{attribute 'conditionalshow'}
FUNCTION_BLOCK FB_GantryXYZ EXTENDS FB_PackML_BaseModule
VAR
    // Sub module definitions here
	RecipeBuilder	:FB_RecipeBuilderWings;

	
	// List of sub modules
    ipSubModules_Init : ARRAY[1..Parameters_PackML_Base.MAX_NO_OF_SUBMODULES] OF I_PackML_BaseModule := [];

    // Component definitions here
    AxisX : FB_Component_BasicAxis := (Name := 'AxisX');
    AxisY : FB_Component_BasicAxis := (Name := 'AxisY');
    AxisZ : FB_Component_BasicAxis := (Name := 'AxisZ');
    CylinderCuttingY : FB_CylinderCutY := (Name := 'Cylinder Y');
	CylinderCuttingX : FB_CylinderCutX := (Name := 'Cylinder X');
	

    // Alarms for this module
    GantryAlarms : ARRAY[1..GANTRY_ALARM_COUNT] OF FB_TcAlarm;
	
    // Properties
    _HomingStepX :			INT;
    _HomingStepY :			INT;
    _HomingStepZ :			INT;

	_ProgramIdRequested :   E_RecipeID;
	_CurrentSpeed: 			LREAL;
	
	//Segments
	SegmentGrooves       : ARRAY[1..32] OF ST_CutSegment;
    SegmentsToGroove     : INT;          // Ile odcinków
    iSegmentsToGroove    : INT;          // Indeks aktualnego odcinka
    
    
	//Segments Cut Y
	SegmentCutY      	 : ARRAY[1..32] OF ST_CutSegment;
    SegmentsToCutY       : INT;          // Ile odcinków
    iSegmentsToCutY      : INT;          // Indeks aktualnego odcinka
	
	//Segments Cut X
	SegmentCutX      	 : ARRAY[1..32] OF ST_CutSegment;
    SegmentsToCutX       : INT;          // Ile odcinków
    iSegmentsToCutX      : INT;          // Indeks aktualnego odcinka

	//Sequencers
	OrchestratorStep :			INT := 0;
	ExecutorStep :				INT := 0;
	
	GantryXYZ_HMI : ST_GantryXYZ_HMI;
	
	//Test
	fbHomeStratX : FB_Homing_StandardNC;
    fbHomeStratY : FB_Homing_StandardNC;
    fbHomeStratZ : FB_Homing_StandardNC;
	
END_VAR

VAR PERSISTENT
	_CuttingSpeedX			:REAL;
	_CuttingSpeedY			:REAL;
	_CuttingIdleTime		:REAL;
	_CuttingOverpass		:REAL;
	_CutterXOffsetX			:REAL;
	_CutterXOffsetY			:REAL;
	_CutterYOffsetX			:REAL;
	_CutterYOffsetY			:REAL;	
    _GrooveDepthZ 			:REAL;
	_GroovingSpeedX 		:REAL;
	_GroovingSpeedY 		:REAL;
	_GroovingSpeedZ 		:REAL;
	_GroovingIdleTime 		:REAL;
    _GroovingOverpass 		:REAL;
    _PanelFrontWidth 		:REAL;
    _PanelHeight 			:REAL;
    _RailHeightCorrection	:REAL;
    _RapidSpeedX 			:REAL;
    _RapidSpeedY 			:REAL;
    _RapidSpeedZ 			:REAL;
	_GlobalOffset 			:INT;
END_VAR

VAR CONSTANT
    GANTRY_ALARM_COUNT : 	INT := 5;
END_VAR


METHOD PROTECTED Aborting
VAR
	i				: UDINT;
	SubModulesReady : BOOL := TRUE;
END_VAR
CASE _CurrentMode OF

	//=================================PRODUCTION MODE==================================
	E_PMLUnitMode.ePMLUnitMode_Production:
CASE SequenceState OF
    0:
        NoStateTasksToComplete := FALSE;
        SequenceState          := SequenceState + 10;
    10:
		AxisX.Disable();
		AxisY.Disable();
		AxisZ.Disable();

		IO.SpindleEnable := FALSE;
		IO.CoolingEnable := FALSE;
		
		CylinderCuttingX.Retract();
		CylinderCuttingY.Retract();

		THIS^.HomingStepX := 0;
		THIS^.HomingStepY := 0;
		THIS^.HomingStepZ := 0;
		OrchestratorStep := 0;
		ExecutorStep := 0;
		
		//test
		fbHomeStratX.Abort();
        fbHomeStratY.Abort();
        fbHomeStratZ.Abort();
		
		SequenceState := SequenceState + 10;
		
		
	20:

		StateTasksComplete := TRUE;
		SUPER^.Aborting();
END_CASE

	//=================================MAINTENANCE & MANUAL MODE==================================
	E_PMLUnitMode.ePMLUnitMode_Maintenance, E_PMLUnitMode.ePMLUnitMode_Manual:

	CASE SequenceState OF
    
	0:
        NoStateTasksToComplete := FALSE;
        SequenceState          := SequenceState + 10;
    
	10:
		AxisX.Disable();
		AxisY.Disable();
		AxisZ.Disable();
		
		IO.CoolingEnable := FALSE;
		IO.SpindleEnable := FALSE;
		THIS^.HomingStepX := 0;
		THIS^.HomingStepY := 0;
		THIS^.HomingStepZ := 0;
		OrchestratorStep := 0;
		SequenceState := SequenceState + 10;
	
	20:
		StateTasksComplete := TRUE;
		SUPER^.Aborting();
	END_CASE
	

	END_CASE
END_METHOD

METHOD BuildSegments_Arona : BOOL
//  Start → Stop, Milling Segments
SegmentsToGroove := 4;

SegmentGrooves[1].Start.X := 500;
SegmentGrooves[1].Start.Y := 500;
SegmentGrooves[1].Stop.X  := 0;
SegmentGrooves[1].Stop.Y  := 500;

SegmentGrooves[2].Start.X := 500;
SegmentGrooves[2].Start.Y := 0;
SegmentGrooves[2].Stop.X  := 0; 
SegmentGrooves[2].Stop.Y  := 0;

SegmentGrooves[3].Start.X := 500;
SegmentGrooves[3].Start.Y := 500;
SegmentGrooves[3].Stop.X  := 500;
SegmentGrooves[3].Stop.Y  := 0;

SegmentGrooves[4].Start.X := 0;
SegmentGrooves[4].Start.Y := 500;
SegmentGrooves[4].Stop.X  := 0;
SegmentGrooves[4].Stop.Y  := 0;

//  Start → Stop, CutY Segments
SegmentsToCutY := 2;

SegmentCutY[1].Start.X := 0; 
SegmentCutY[1].Start.Y := 500;  
SegmentCutY[1].Stop.X  := 0; 
SegmentCutY[1].Stop.Y  := 0;
SegmentCutY[2].Start.X := 500; 
SegmentCutY[2].Start.Y := 500;  
SegmentCutY[2].Stop.X  := 500; 
SegmentCutY[2].Stop.Y  := 0;

SegmentsToCutX := 2;

SegmentCutX[1].Start.X := 500; 
SegmentCutX[1].Start.Y := 500;  
SegmentCutX[1].Stop.X  := 500; 
SegmentCutX[1].Stop.Y  := 0;
SegmentCutX[2].Start.X := 0; 
SegmentCutX[2].Start.Y := 500;  
SegmentCutX[2].Stop.X  := 0; 
SegmentCutX[2].Stop.Y  := 0;



BuildSegments_Arona := TRUE;
END_METHOD

METHOD BuildSegments_BorgoFlaps : BOOL
VAR_INST
	TotalY 		:REAL;
	TotalX  	:REAL;
	ShorterY  	:REAL;
	ShorterX  	:REAL;
END_VAR
//Natural language parameters;
//TotalY := PanelFrontLength + 2 * _PanelHeight;
TotalX := PanelFrontWidth + 2 * _PanelHeight;
ShorterY := TotalY - _PanelHeight;
ShorterX := TotalX - _PanelHeight;


SegmentsToGroove := 4;

///////////////
SegmentGrooves[1].Start.X := TotalX;
SegmentGrooves[1].Stop.X := 0;

SegmentGrooves[1].Start.Y := ShorterY;
SegmentGrooves[1].Stop.Y := ShorterY;

/////////////
SegmentGrooves[2].Start.Y := TotalY;
SegmentGrooves[2].Stop.Y := 0;

SegmentGrooves[2].Start.X := _PanelHeight;
SegmentGrooves[2].Stop.X := _PanelHeight;

///////////////
SegmentGrooves[3].Start.X := 0;
SegmentGrooves[3].Stop.X :=  TotalX; 

SegmentGrooves[3].Start.Y := _PanelHeight;
SegmentGrooves[3].Stop.Y :=  _PanelHeight;

//////////////
SegmentGrooves[4].Start.X := ShorterX;
SegmentGrooves[4].Stop.X := ShorterX;

SegmentGrooves[4].Start.Y := 0;
SegmentGrooves[4].Stop.Y := TotalY;





//  Start → Stop, CutY Segments
SegmentsToCutY := 0;

SegmentsToCutX := 0;

BuildSegments_BorgoFlaps := TRUE;
END_METHOD

METHOD BuildSegments_BorgoWings : BOOL
VAR_INST
	TotalY 		:REAL;
	TotalX  	:REAL;
	ShorterY  	:REAL;
	ShorterX  	:REAL;
END_VAR

//We cut here BorgoWings it means, panel will be installed on wings
// It means we have to make flaps shorter
//Natural language parameters;
//TotalY := PanelFrontLength + 2 * _PanelHeight;
TotalX := PanelFrontWidth + 2 * _PanelHeight;
ShorterY := TotalY - _PanelHeight;
ShorterX := TotalX - _PanelHeight;



//  Start → Stop, Milling Segments
SegmentsToGroove := 4;

///////////////
SegmentGrooves[1].Start.X := TotalX;
SegmentGrooves[1].Stop.X := 0;

SegmentGrooves[1].Start.Y := ShorterY;
SegmentGrooves[1].Stop.Y := ShorterY;

///////////////
SegmentGrooves[2].Start.X := TotalX;
SegmentGrooves[2].Stop.X :=  0; 

SegmentGrooves[2].Start.Y := _PanelHeight;
SegmentGrooves[2].Stop.Y :=  _PanelHeight;

//////////////
SegmentGrooves[3].Start.X := ShorterX;
SegmentGrooves[3].Stop.X := ShorterX;

SegmentGrooves[3].Start.Y := TotalY;
SegmentGrooves[3].Stop.Y := 0;

/////////////
SegmentGrooves[4].Start.Y := TotalY;
SegmentGrooves[4].Stop.Y := 0;

SegmentGrooves[4].Start.X := _PanelHeight;
SegmentGrooves[4].Stop.X := _PanelHeight;


////////////
// Cut X //
///////////
SegmentsToCutX := 6;

//Short Box Segments
SegmentCutX[1].Start.X := TotalX + _CuttingOverpass;
SegmentCutX[1].Stop.X  := ShorterX;

SegmentCutX[1].Start.Y := ShorterY;
SegmentCutX[1].Stop.Y  := ShorterY;

///////////////
SegmentCutX[2].Start.X := _PanelHeight;
SegmentCutX[2].Stop.X  := -_CuttingOverpass;

SegmentCutX[2].Start.Y := ShorterY;
SegmentCutX[2].Stop.Y  := ShorterY;

///////////////
SegmentCutX[3].Start.X := TotalX + _CuttingOverpass;
SegmentCutX[3].Stop.X := ShorterX;

SegmentCutX[3].Start.Y := _PanelHeight;
SegmentCutX[3].Stop.Y := _PanelHeight;

///////////////
SegmentCutX[4].Start.X := _PanelHeight;
SegmentCutX[4].Stop.X :=  -_CuttingOverpass;

SegmentCutX[4].Start.Y := _PanelHeight;
SegmentCutX[4].Stop.Y := _PanelHeight;

//Panel Dimensions Shorter Flaps


SegmentCutX[5].Start.X := TotalX + _CuttingOverpass;
SegmentCutX[5].Stop.X  := - _CuttingOverpass;

SegmentCutX[5].Start.Y := TotalY - _RailHeightCorrection;
SegmentCutX[5].Stop.Y  := TotalY - _RailHeightCorrection;

///////////////
SegmentCutX[6].Start.X := TotalX + _CuttingOverpass;
SegmentCutX[6].Stop.X  := - _CuttingOverpass;

SegmentCutX[6].Start.Y := _RailHeightCorrection;
SegmentCutX[6].Stop.Y  := _RailHeightCorrection;


////////////
// Cut Y //
///////////

SegmentsToCutY := 6;

//Short Box Segments
SegmentCutY[1].Start.X := ShorterX;
SegmentCutY[1].Stop.X  := ShorterX;

SegmentCutY[1].Start.Y := TotalY + _CuttingOverpass;
SegmentCutY[1].Stop.Y  := ShorterY;

///////////////
SegmentCutY[2].Start.X := _PanelHeight;
SegmentCutY[2].Stop.X  := _PanelHeight;

SegmentCutY[2].Start.Y := TotalY + _CuttingOverpass;
SegmentCutY[2].Stop.Y  := ShorterY;

///////////////
SegmentCutY[3].Start.X := ShorterX;
SegmentCutY[3].Stop.X  := ShorterX;

SegmentCutY[3].Start.Y := _PanelHeight;
SegmentCutY[3].Stop.Y  := -_CuttingOverpass;

///////////////
SegmentCutY[4].Start.X := _PanelHeight;
SegmentCutY[4].Stop.X  := _PanelHeight;

SegmentCutY[4].Start.Y := _PanelHeight;
SegmentCutY[4].Stop.Y  := -_CuttingOverpass;

//Panel Dimensions
SegmentCutY[5].Start.X := TotalX;
SegmentCutY[5].Stop.X  := TotalX;

SegmentCutY[5].Start.Y := TotalY + _CuttingOverpass;
SegmentCutY[5].Stop.Y  := -_CuttingOverpass;
///////////////
SegmentCutY[6].Start.X := 0;
SegmentCutY[6].Stop.X  := 0;

SegmentCutY[6].Start.Y := TotalY + _CuttingOverpass;
SegmentCutY[6].Stop.Y  := - _CuttingOverpass;



BuildSegments_BorgoWings := TRUE;
END_METHOD

METHOD BuildSegments_Calibration : BOOL
VAR_INST
	TotalLength :REAL;
	TotalWidth  :REAL;
	WingHeight  :REAL;
	FlapHeight  :REAL;
END_VAR
//  Start → Stop, Milling Segments
SegmentsToGroove := 4;

SegmentGrooves[1].Start.X := 300;
SegmentGrooves[1].Start.Y := 300;
SegmentGrooves[1].Stop.X  := 50;
SegmentGrooves[1].Stop.Y  := 300;

SegmentGrooves[2].Start.X := 300;
SegmentGrooves[2].Start.Y := 50;
SegmentGrooves[2].Stop.X  := 50; 
SegmentGrooves[2].Stop.Y  := 50;

SegmentGrooves[3].Start.X := 300;
SegmentGrooves[3].Start.Y := 300;
SegmentGrooves[3].Stop.X  := 300;
SegmentGrooves[3].Stop.Y  := 50;

SegmentGrooves[4].Start.X := 50;
SegmentGrooves[4].Start.Y := 300;
SegmentGrooves[4].Stop.X  := 50;
SegmentGrooves[4].Stop.Y  := 50;

//  Start → Stop, CutY Segments
SegmentsToCutY := 2;

SegmentCutY[1].Start.X := 300; 
SegmentCutY[1].Start.Y := 300;  
SegmentCutY[1].Stop.X  := 300; 
SegmentCutY[1].Stop.Y  := 50;

SegmentCutY[2].Start.X := 50; 
SegmentCutY[2].Start.Y := 300;  
SegmentCutY[2].Stop.X  := 50; 
SegmentCutY[2].Stop.Y  := 50;

SegmentsToCutX := 2;

SegmentCutX[1].Start.X := 300;
SegmentCutX[1].Start.Y := 300; 
SegmentCutX[1].Stop.X  := 50;
SegmentCutX[1].Stop.Y  := 300;
                               
SegmentCutX[2].Start.X := 300;
SegmentCutX[2].Start.Y := 50; 
SegmentCutX[2].Stop.X  := 50; 
SegmentCutX[2].Stop.Y  := 50;

BuildSegments_Calibration := TRUE;
END_METHOD

METHOD PROTECTED Clearing
VAR
	i				: UDINT;
	SubModulesReady : BOOL := TRUE;
END_VAR

VAR_INST
	//SoEResetAxis1 : FB_SoEReset;
	//ResetAxis1 :	MC_Reset;
END_VAR
CASE SequenceState OF
    0:
        NoStateTasksToComplete := FALSE;
        SequenceState          := SequenceState + 10;
    10:
		//Reset any alarms that get latched
//		GantryAlarms[E_Gantry.AlarmMessage].Clear(0,0);		
//		GantryAlarms[E_Gantry.InfoMessage].Clear(0,0);
//		GantryAlarms[E_Gantry.InitReferenceEvent].Clear(0,0);
//		GantryAlarms[E_Gantry.StartTimeout].Clear(0,0);
//		GantryAlarms[E_Gantry.WarnMessage].Clear(0,0);
		THIS^.HomingStepX := 0;
		THIS^.HomingStepY := 0;
		THIS^.HomingStepZ := 0;
		AxisX.Reset();
		AxisY.Reset();
		AxisZ.Reset();

		SequenceState := SequenceState + 10;
	20:
	
		SequenceState := SequenceState + 10;
	30: 

		IF ResetSafety() THEN
			SequenceState := SequenceState + 10;		
		END_IF	
    40:

        // Enable here
		// AxisX.Enable();
		// AxisY.Enable();
		// AxisZ.Enable();

        // Check enabled here
		// IF AxisX.Enabled AND AxisY.Enabled AND AxisZ.Enabled THEN
			// SequenceState := SequenceState + 10;
		// END_IF
		
		SequenceState := SequenceState + 10;
		
    50:
        StateTasksComplete := TRUE;
		
END_CASE

SUPER^.Clearing();
END_METHOD

// This method contains code which will execute when this PackML module is in the Completing state
METHOD PROTECTED Completing
VAR
	i				: UDINT;
	SubModulesReady : BOOL := TRUE;
END_VAR

// This method is called as required by <c>StateControl()</c>
CASE _CurrentMode OF

	//=================================PRODUCTION MODE==================================
	E_PMLUnitMode.ePMLUnitMode_Production:
		CASE SequenceState OF
		0:
			NoStateTasksToComplete := FALSE;
			SequenceState          := SequenceState + 10;
		10:
			SequenceState := SequenceState + 10;
		20:
			StateTasksComplete := TRUE;
			SUPER^.Completing();
	END_CASE

	//=================================MAINTENANCE & MANUAL MODE==================================
	E_PMLUnitMode.ePMLUnitMode_Maintenance, E_PMLUnitMode.ePMLUnitMode_Manual:
			

		SUPER^.Completing();

END_CASE
END_METHOD

METHOD PROTECTED CreateEvents
VAR_INPUT
END_VAR
// Add your event creation here
F_CreateAllEventsInClass(Alarms     := GantryAlarms,
                         ClassSize  := SIZEOF(TC_EVENTS.Gantry),
                         pInitEvent := ADR(TC_EVENTS.Gantry.InitReferenceEvent),
                         Prefix     := _Name);

// Super call to base
SUPER^.CreateEvents();
END_METHOD

PROPERTY CurrentSpeed : LREAL
GET
CurrentSpeed := _CurrentSpeed;
END_GET
END_PROPERTY

PROPERTY PUBLIC CutterXOffsetX : REAL
GET
CutterXOffsetX := _CutterXOffsetX;
END_GET
SET
_CutterXOffsetX := CutterXOffsetX;
END_SET
END_PROPERTY

PROPERTY PUBLIC CutterXOffsetY : REAL
GET
CutterXOffsetY := _CutterXOffsetY;
END_GET
SET
_CutterXOffsetY := CutterXOffsetY;
END_SET
END_PROPERTY

PROPERTY PUBLIC CutterYOffsetX : REAL
GET
CutterYOffsetX := _CutterYOffsetX;
END_GET
SET
_CutterYOffsetX := CutterYOffsetX;
END_SET
END_PROPERTY

PROPERTY PUBLIC CutterYOffsetY : REAL
GET
CutterYOffsetY := _CutterYOffsetY;
END_GET
SET
_CutterYOffsetY := CutterYOffsetY;
END_SET
END_PROPERTY

PROPERTY PUBLIC CuttingIdleTime : REAL
GET
CuttingIdleTime := _CuttingIdleTime;
END_GET
SET
_CuttingIdleTime := CuttingIdleTime;
END_SET
END_PROPERTY

PROPERTY PUBLIC CuttingOverpass : REAL
GET
CuttingOverpass := _CuttingOverpass;
END_GET
SET
_CuttingOverpass := CuttingOverpass;
END_SET
END_PROPERTY

PROPERTY PUBLIC CuttingSpeedX : REAL
GET
CuttingSpeedX := _CuttingSpeedX;
END_GET
SET
_CuttingSpeedX := CuttingSpeedX;
END_SET
END_PROPERTY

PROPERTY PUBLIC CuttingSpeedY : REAL
GET
CuttingSpeedY := _CuttingSpeedY;
END_GET
SET
_CuttingSpeedY := CuttingSpeedY;
END_SET
END_PROPERTY

METHOD CyclicLogic
VAR_INPUT
END_VAR
IF NOT _InitComplete THEN
    _InitComplete := Initialize();
    RETURN;
END_IF

//aaa(
//	Axis := AxisY.Axis , 
//	Execute := TRUE , 
//	ParameterNumber := MC_AxisParameter.AxisMinSoftPosLimit , 
//	Value := -66, 
//	 );
	 
	 
_CurrentSpeed := SQRT( AxisX.SetVelocity*AxisX.SetVelocity + AxisY.SetVelocity*AxisY.SetVelocity + AxisZ.SetVelocity*AxisZ.SetVelocity );


SUPER^.CyclicLogic();

fbHomeStratX.bSensorInput := IO.ProximitySensorX;
fbHomeStratY.bSensorInput := IO.ProximitySensorY;
fbHomeStratZ.bSensorInput := IO.ProximitySensorZ;

fbHomeStratX.CyclicLogic();
fbHomeStratY.CyclicLogic();
fbHomeStratZ.CyclicLogic();

//Set the current alarm severity for this module
_CurrentAlarmSeverity := F_GetMaxSeverityRaised(Alarms := GantryAlarms, CurrentSeverity := _CurrentAlarmSeverity);

//Simulate Alarm Messaging
END_METHOD

METHOD PROTECTED Execute
CASE _CurrentMode OF

	//=================================PRODUCTION MODE==================================
	E_PMLUnitMode.ePMLUnitMode_Production:
		CASE SequenceState OF
			0:
				NoStateTasksToComplete := FALSE;
				SequenceState := SequenceState + 5;
			5:
				AxisX.WriteParameter(MC_AxisParameter.AxisMinSoftPosLimit, -20);	 
				AxisX.WriteParameter(MC_AxisParameter.AxisMaxSoftPosLimit, 1200);
		
				AxisY.WriteParameter(MC_AxisParameter.AxisMinSoftPosLimit, -20);	 
				AxisY.WriteParameter(MC_AxisParameter.AxisMaxSoftPosLimit, 2300);
		
				AxisZ.WriteParameter(MC_AxisParameter.AxisMinSoftPosLimit, -20);	 
				AxisZ.WriteParameter(MC_AxisParameter.AxisMaxSoftPosLimit, 100);	
				SequenceState := SequenceState + 5;
			10:
					
				IF MachiningOrchestrator() THEN
					SequenceState := SequenceState + 10;
				END_IF
				
			
			
//				CASE GVL_HMI.ProgramToCut OF
					
//					0:
//					IF CutBorgoFlaps() THEN
//						SequenceState := SequenceState + 10;
//					END_IF
					
//					1:
//					IF CutBorgoWings() THEN
//						SequenceState := SequenceState + 10;
//					END_IF
					
//					2:
//					IF CutOrchestrator() THEN
//						SequenceState := SequenceState + 10;
//					END_IF
					
//				END_CASE
			
								
			20:		
				StateTasksComplete := TRUE;
				StateComplete();
			END_CASE

	//=================================MAINTENANCE & MANUAL MODE==================================
	E_PMLUnitMode.ePMLUnitMode_Maintenance, E_PMLUnitMode.ePMLUnitMode_Manual:
		;
END_CASE
END_METHOD

METHOD ExecuteSegmentsCutX : BOOL
CASE ExecutorStep OF

// -------- Inicjalizacja pierwszego segmentu --------
0:
IF AxisX.Enable() AND AxisY.Enable() AND AxisZ.Enable() THEN
			 Trace('SegmentExecutionX');
			 
			 
    IF SegmentsToCutX <= 0 THEN
        // Nie ma czego ciąć
        ExecuteSegmentsCutX := TRUE;
        RETURN;
    END_IF;

    // Jednorazowe nastawy:
    AxisX.Acceleration := 500;   AxisX.Deceleration := 8000;
    AxisY.Acceleration := 500;   AxisY.Deceleration := 8000;
    AxisZ.Acceleration := 500;   AxisZ.Deceleration := 8000;

    AxisX.Velocity := _RapidSpeedX;
    AxisY.Velocity := _RapidSpeedY;
    AxisZ.Velocity := _RapidSpeedZ;

	iSegmentsToCutX := 0;
	
	IF NOT AxisX.Busy AND NOT AxisY.Busy AND NOT AxisZ.Busy THEN
		iSegmentsToCutX := iSegmentsToCutX + 1;
		ExecutorStep := 10;
	END_IF	 
   
END_IF

10:
    AxisX.MoveAbsolute(SegmentCutX[iSegmentsToCutX].Start.X + _CutterXOffsetX + _GlobalOffset, 0);
    AxisY.MoveAbsolute(SegmentCutX[iSegmentsToCutX].Start.Y + _CutterXOffsetY + _GlobalOffset, 0);
    ExecutorStep := 20;

20: // czekamy na pozycję XY
    IF AxisX.InPosition AND AxisY.InPosition THEN 
        ExecutorStep := 30;
    END_IF


30:
	CylinderCuttingX.Extend();
	ExecutorStep := 40;

40: 
	IF CylinderCuttingX.Extended THEN
	AxisX.Velocity := _CuttingSpeedX;
	AxisY.Velocity := _CuttingSpeedY;
	ExecutorStep := 50;
    END_IF
		
	
50:
   	IF SequenceTimerSeconds(_CuttingIdleTime) THEN
		ExecutorStep := 60;
	END_IF

// -------- Cięcie XY do końca odcinka --------
60:
    AxisX.MoveAbsolute(SegmentCutX[iSegmentsToCutX].Stop.X + _CutterXOffsetX + _GlobalOffset, 0);
    AxisY.MoveAbsolute(SegmentCutX[iSegmentsToCutX].Stop.Y + _CutterXOffsetY + _GlobalOffset, 0);
    ExecutorStep := 70;

70: // czekamy na koniec cięcia
    IF AxisX.InPosition AND AxisY.InPosition THEN
        ExecutorStep := 80;
    END_IF

// -------- Retrakt Z i przygotowanie następnego --------
80:
	CylinderCuttingX.Retract();
		ExecutorStep := 85;
	
85: 
	IF CylinderCuttingX.Retracted THEN
		 iSegmentsToCutX := iSegmentsToCutX + 1; 
		 ExecutorStep := 90;
	END_IF	

90:
    IF SequenceTimerSeconds(_CuttingIdleTime) THEN
        AxisX.Velocity := _RapidSpeedX;
        AxisY.Velocity := _RapidSpeedY;

        
        IF iSegmentsToCutX > SegmentsToCutX THEN
            ExecutorStep := 1000; // koniec
        ELSE
            ExecutorStep := 10;   // następny odcinek
        END_IF
    END_IF

// -------- Zakończenie --------
1000:
	ExecutorStep := 0;
	Trace('SegmentExecutionX-FINISHED');
    ExecuteSegmentsCutX := TRUE;
END_CASE
END_METHOD

METHOD ExecuteSegmentsCutY : BOOL
CASE ExecutorStep OF

// -------- Inicjalizacja pierwszego segmentu --------
0:
IF AxisX.Enable() AND AxisY.Enable() AND AxisZ.Enable() THEN
			 Trace('SegmentExecutionY');
			 
			 
    IF SegmentsToCutY <= 0 THEN
        // Nie ma czego ciąć
        ExecuteSegmentsCutY := TRUE;
        RETURN;
    END_IF;

    // Jednorazowe nastawy:
    AxisX.Acceleration := 500;   AxisX.Deceleration := 8000;
    AxisY.Acceleration := 500;   AxisY.Deceleration := 8000;
    AxisZ.Acceleration := 500;   AxisZ.Deceleration := 8000;

    AxisX.Velocity := _RapidSpeedX;
    AxisY.Velocity := _RapidSpeedY;
    AxisZ.Velocity := _RapidSpeedZ;

	iSegmentsToCutY := 0;
	
	IF NOT AxisX.Busy AND NOT AxisY.Busy AND NOT AxisZ.Busy THEN
		iSegmentsToCutY := iSegmentsToCutY + 1;
		ExecutorStep := 10;
	END_IF	 
   
END_IF

10:
    AxisX.MoveAbsolute(SegmentCutY[iSegmentsToCutY].Start.X + _CutterYOffsetX + _GlobalOffset, 0);
    AxisY.MoveAbsolute(SegmentCutY[iSegmentsToCutY].Start.Y + _CutterYOffsetY + _GlobalOffset, 0);
    ExecutorStep := 20;

20: // czekamy na pozycję XY
    IF AxisX.InPosition AND AxisY.InPosition THEN 
        ExecutorStep := 30;
    END_IF


30:
	CylinderCuttingY.Extend();
	ExecutorStep := 40;

40: 
	IF CylinderCuttingY.Extended THEN
    //IF IO.PistonSensorCutY THEN
	AxisX.Velocity := _CuttingSpeedX;
	AxisY.Velocity := _CuttingSpeedY;
	ExecutorStep := 50;
    END_IF
		
	
50:
   	IF SequenceTimerSeconds(_CuttingIdleTime) THEN
		ExecutorStep := 60;
	END_IF

// -------- Cięcie XY do końca odcinka --------
60:
    AxisX.MoveAbsolute(SegmentCutY[iSegmentsToCutY].Stop.X + _CutterYOffsetX + _GlobalOffset, 0);
    AxisY.MoveAbsolute(SegmentCutY[iSegmentsToCutY].Stop.Y + _CutterYOffsetY + _GlobalOffset, 0);
    ExecutorStep := 70;

70: // czekamy na koniec cięcia
    IF AxisX.InPosition AND AxisY.InPosition THEN
        ExecutorStep := 80;
    END_IF

// -------- Retrakt Z i przygotowanie następnego --------
80:
	CylinderCuttingY.Retract();
//	IO.PistonValveCutY := FALSE;
		ExecutorStep := 85;
	
85: 
	IF CylinderCuttingY.Retracted THEN
	//IF NOT IO.PistonSensorCutY  THEN
		 iSegmentsToCutY := iSegmentsToCutY + 1; 
		 ExecutorStep := 90;
	END_IF	

90:
    IF SequenceTimerSeconds(_CuttingIdleTime) THEN
        AxisX.Velocity := _RapidSpeedX;
        AxisY.Velocity := _RapidSpeedY;

        
        IF iSegmentsToCutY > SegmentsToCutY THEN
            ExecutorStep := 1000; // koniec
        ELSE
            ExecutorStep := 10;   // następny odcinek
        END_IF
    END_IF

// -------- Zakończenie --------
1000:
	ExecutorStep := 0;
	Trace('SegmentExecutionYFINISHED');
    ExecuteSegmentsCutY := TRUE;
END_CASE
END_METHOD

METHOD ExecuteSegmentsGroove : BOOL
VAR_INST
iPass : INT;
currentDepth : LREAL;
g1, g2, g3, g4, g5 : LREAL;
v1, v2, v3, v4, v5 : LREAL;
END_VAR
CASE ExecutorStep OF

    // -------- Inicjalizacja --------
    0:
        // Konfiguracja głębokości (g) i mnożników prędkości (v)
        g1 := 3.5; 
        g2 := 3.5; 
        g3 := 1.5; 
        g4 := 0.0;
        g5 := 0.0; // Ostatnie przejście na pełną głębokość

        v1 := 1.0;
        v2 := 1.0;
        v3 := 1.0;
        v4 := 0.4;
        v5 := 0.4; // Np. wolniej na wykończenie

        IF AxisX.Enable() AND AxisY.Enable() AND AxisZ.Enable() THEN
            
            IF iSegmentsToGroove = 0 THEN 
                Trace(Message:= 'Step 0: Start Initialization (5 Passes Mode)'); 
            END_IF;

            IF SegmentsToGroove <= 0 THEN
                Trace(Message:= 'Step 0: No segments, going to 1000');
                IO.SpindleEnable := FALSE;
                ExecutorStep := 1000;
                RETURN;
            END_IF;

            // Jednorazowe nastawy dynamiki
            AxisX.Acceleration := 500; AxisX.Deceleration := 8000;
            AxisY.Acceleration := 500; AxisY.Deceleration := 8000;
            AxisZ.Acceleration := 500; AxisZ.Deceleration := 8000;

            AxisX.Velocity := _RapidSpeedX;
            AxisY.Velocity := _RapidSpeedY;
            AxisZ.Velocity := _RapidSpeedZ;

            IO.SpindleEnable := TRUE;
            IO.CoolingEnable := FALSE;

            iSegmentsToGroove := 1;
            //od którego poziomu zaczynac, ostroznie
			iPass := 4; 

            IF NOT AxisX.Busy AND NOT AxisY.Busy AND NOT AxisZ.Busy THEN
                Trace(Message:= 'Step 0: Axes ready, going to 10');
                ExecutorStep := 10;
            END_IF
        END_IF;

    10: 
        Trace(Message:= CONCAT('Step 10: Rapid to Start XY. Pass: ', TO_STRING(iPass)));
        
        AxisX.MoveAbsolute(SegmentGrooves[iSegmentsToGroove].Start.X + _GlobalOffset, 0);
        AxisY.MoveAbsolute(SegmentGrooves[iSegmentsToGroove].Start.Y + _GlobalOffset, 0);
        ExecutorStep := 20;

    20: 
        IF AxisX.InPosition AND AxisY.InPosition THEN
            IO.SpindleEnable := TRUE;
            IO.CoolingEnable := TRUE;
            AxisZ.Velocity := _GroovingSpeedZ;
            ExecutorStep := 30;
        END_IF;

    30: 
        // Wybór głębokości dla 5 przejść
        CASE iPass OF
            1: currentDepth := _GrooveDepthZ - g1;
            2: currentDepth := _GrooveDepthZ - g2;
            3: currentDepth := _GrooveDepthZ - g3;
            4: currentDepth := _GrooveDepthZ - g4;
            5: currentDepth := _GrooveDepthZ - g5;
        ELSE
            currentDepth := _GrooveDepthZ;
        END_CASE;

        Trace(Message:= CONCAT('Step 30: Pass ', CONCAT(TO_STRING(iPass), CONCAT(' Moving Z to: ', TO_STRING(currentDepth)))));

        AxisZ.MoveAbsolute(currentDepth, 0);
        ExecutorStep := 40;

    40: 
        IF AxisZ.InPosition THEN
            // Wybór prędkości posuwu dla 5 przejść
            CASE iPass OF
                1:
                    AxisX.Velocity := _GroovingSpeedX * v1;
                    AxisY.Velocity := _GroovingSpeedY * v1;
                2: 
                    AxisX.Velocity := _GroovingSpeedX * v2;
                    AxisY.Velocity := _GroovingSpeedY * v2;
                3: 
                    AxisX.Velocity := _GroovingSpeedX * v3;
                    AxisY.Velocity := _GroovingSpeedY * v3;
                4: 
                    AxisX.Velocity := _GroovingSpeedX * v4;
                    AxisY.Velocity := _GroovingSpeedY * v4;
                5: 
                    AxisX.Velocity := _GroovingSpeedX * v5;
                    AxisY.Velocity := _GroovingSpeedY * v5;
            END_CASE;

            ExecutorStep := 50;
        END_IF;

    50: 
        IF SequenceTimerSeconds(_GroovingIdleTime) THEN
            ExecutorStep := 60;
        END_IF;

    60: 
        Trace(Message:= 'Step 60: Cutting Move to Stop XY');
        
        AxisX.MoveAbsolute(SegmentGrooves[iSegmentsToGroove].Stop.X + _GlobalOffset, 0);
        AxisY.MoveAbsolute(SegmentGrooves[iSegmentsToGroove].Stop.Y + _GlobalOffset, 0);
        ExecutorStep := 70;

    70: 
        IF AxisX.InPosition AND AxisY.InPosition AND AxisZ.InPosition THEN
            // Sprawdzamy czy to ostatnie przejście (teraz 5)
            IF iPass = 5 THEN
                Trace(Message:= 'Step 70: Pass 5 (Final) -> Going to Return Path');
                ExecutorStep := 74;
            ELSE
                Trace(Message:= 'Step 70: Intermediate Pass -> Lifting Z');
                AxisZ.Velocity := _RapidSpeedZ;
                ExecutorStep := 80;
            END_IF;
        END_IF;
        
    74:
        IF SequenceTimerSeconds(0.5) THEN
            ExecutorStep := 75;
        END_IF;

    75: 
        Trace(Message:= 'Step 75: Cleaning Return (Z stays down)');
        AxisX.MoveAbsolute(SegmentGrooves[iSegmentsToGroove].Start.X + _GlobalOffset, 0);
        AxisY.MoveAbsolute(SegmentGrooves[iSegmentsToGroove].Start.Y + _GlobalOffset, 0);
        ExecutorStep := 76;
        
    76: 
        IF AxisX.InPosition AND AxisY.InPosition THEN
            AxisZ.Velocity := _RapidSpeedZ;
            ExecutorStep := 80; 
        END_IF;

    80: 
        Trace(Message:= 'Step 80: Lifting Z to Safe 0');
        AxisZ.MoveAbsolute(0, 0);
        ExecutorStep := 90;

    90: 
        IF AxisZ.InPosition THEN
            ExecutorStep := 100;
        END_IF;

    100: 
        IF SequenceTimerSeconds(_GroovingIdleTime) THEN
            
            AxisX.Velocity := _RapidSpeedX;
            AxisY.Velocity := _RapidSpeedY;
            
            iSegmentsToGroove := iSegmentsToGroove + 1;

            // Logika zmiany przejścia lub zakończenia
            IF iSegmentsToGroove > SegmentsToGroove THEN
                IF iPass < 5 THEN
                    Trace(Message:= CONCAT('Step 100: Pass ', CONCAT(TO_STRING(iPass), ' finished. Moving to next pass.')));
                    iPass := iPass + 1;       
                    iSegmentsToGroove := 1;   
                    ExecutorStep := 10;       
                ELSE
                    Trace(Message:= 'Step 100: ALL 5 PASSES DONE. Finishing.');
                    IO.SpindleEnable := FALSE; 
                    IO.CoolingEnable := FALSE; 
                    ExecutorStep := 1000;      
                END_IF;
            ELSE
                ExecutorStep := 10;
            END_IF;
        END_IF;

    1000:
        Trace(Message:= 'Step 1000: FINISH');
        ExecutorStep := 0;
        ExecuteSegmentsGroove := TRUE;

END_CASE;
END_METHOD

PROPERTY PUBLIC GlobalOffset : INT
GET
GlobalOffset := _GlobalOffset;
END_GET
SET
_GlobalOffset := GlobalOffset;
END_SET
END_PROPERTY

PROPERTY PUBLIC GrooveDepthZ : REAL
GET
GrooveDepthZ := _GrooveDepthZ;
END_GET
SET
_GrooveDepthZ := GrooveDepthZ;
END_SET
END_PROPERTY

PROPERTY PUBLIC GroovingIdleTime : REAL
GET
GroovingIdleTime := _GroovingIdleTime;
END_GET
SET
_GroovingIdleTime := GroovingIdleTime;
END_SET
END_PROPERTY

PROPERTY PUBLIC GroovingOverpass : REAL
GET
GroovingOverpass := _GroovingOverpass;
END_GET
SET
_GroovingOverpass := GroovingOverpass;
END_SET
END_PROPERTY

PROPERTY PUBLIC GroovingSpeedX : REAL
GET
GroovingSpeedX := _GroovingSpeedX;
END_GET
SET
_GroovingSpeedX := GroovingSpeedX;
END_SET
END_PROPERTY

PROPERTY PUBLIC GroovingSpeedY : REAL
GET
GroovingSpeedY := _GroovingSpeedY;
END_GET
SET
_GroovingSpeedY := GroovingSpeedY;
END_SET
END_PROPERTY

PROPERTY PUBLIC GroovingSpeedZ : REAL
GET
GroovingSpeedZ := _GroovingSpeedZ;
END_GET
SET
_GroovingSpeedZ := GroovingSpeedZ;
END_SET
END_PROPERTY

// Provides interlocks for HMI control and updates HMI status information for this module
//Only in this place HMI input can overwrite internal data 
METHOD PROTECTED HMICommunication
// This method is called cyclically by CyclicLogic()
SUPER^.HMICommunication();

_CutterXOffsetX       := GantryXYZ_HMI.Config.CutterXOffsetX;
_CutterXOffsetY       := GantryXYZ_HMI.Config.CutterXOffsetY;
_CutterYOffsetX       := GantryXYZ_HMI.Config.CutterYOffsetX;
_CutterYOffsetY       := GantryXYZ_HMI.Config.CutterYOffsetY;
_CuttingSpeedX        := GantryXYZ_HMI.Config.CuttingSpeedX;
_CuttingSpeedY        := GantryXYZ_HMI.Config.CuttingSpeedY;
_CuttingIdleTime      := GantryXYZ_HMI.Config.CuttingIdleTime;
_CuttingOverpass      := GantryXYZ_HMI.Config.CuttingOverpass;
_GrooveDepthZ         := GantryXYZ_HMI.Config.GrooveDepthZ;
_GroovingSpeedX       := GantryXYZ_HMI.Config.GroovingSpeedX;
_GroovingSpeedY       := GantryXYZ_HMI.Config.GroovingSpeedY;
_GroovingSpeedZ       := GantryXYZ_HMI.Config.GroovingSpeedZ;
_ProgramIdRequested   := GantryXYZ_HMI.Command.ProgramIdRequested;
_RapidSpeedX          := GantryXYZ_HMI.Config.RapidSpeedX;
_RapidSpeedY          := GantryXYZ_HMI.Config.RapidSpeedY;
_RapidSpeedZ          := GantryXYZ_HMI.Config.RapidSpeedZ;
_GroovingIdleTime     := GantryXYZ_HMI.Config.GroovingIdleTime;
_GroovingOverpass     := GantryXYZ_HMI.Config.GroovingOverpass;
_GlobalOffset		  := GantryXYZ_HMI.Config.GlobalOffset;

_PanelFrontWidth      := GantryXYZ_HMI.Config.PanelFrontWidht;

_PanelHeight          := GantryXYZ_HMI.Config.PanelHeight;
_RailHeightCorrection := GantryXYZ_HMI.Config.RailHeightCorrection;
END_METHOD

METHOD PROTECTED HMIPermissions
//General Mode Based Monitoring and handling of HMI control
CASE _CurrentMode OF
   
 E_PMLUnitMode.ePMLUnitMode_Production:
        CASE _CurrentState OF
            E_PMLState.ePMLState_Stopped:
				AllowHMIControl(ThisModuleOnly := FALSE);
            E_PMLState.ePMLState_Idle:
				AllowHMIControl(ThisModuleOnly := FALSE);
            E_PMLState.ePMLState_Suspended:
         		AllowHMIControl(ThisModuleOnly := FALSE);
            E_PMLState.ePMLState_Execute:
            	AllowHMIControl(ThisModuleOnly := FALSE); 
            E_PMLState.ePMLState_Aborted:
                AllowHMIControl(ThisModuleOnly := FALSE); 
            E_PMLState.ePMLState_Held:
                AllowHMIControl(ThisModuleOnly := FALSE); 
            E_PMLState.ePMLState_Complete:
          		AllowHMIControl(ThisModuleOnly := FALSE); 
        END_CASE
		
    E_PMLUnitMode.ePMLUnitMode_Manual:
        AllowHMIControl(ThisModuleOnly := FALSE); 
	E_PMLUnitMode.ePMLUnitMode_Maintenance:
        AllowHMIControl(ThisModuleOnly := FALSE); 
END_CASE
END_METHOD

PROPERTY PUBLIC HomingStepX : INT
GET
HomingStepX := _HomingStepX;
END_GET
SET
_HomingStepX := HomingStepX;
END_SET
END_PROPERTY

PROPERTY PUBLIC HomingStepY : INT
GET
HomingStepY := _HomingStepY;
END_GET
SET
_HomingStepY := HomingStepY;
END_SET
END_PROPERTY

PROPERTY PUBLIC HomingStepZ : INT
GET
HomingStepZ := _HomingStepZ;
END_GET
SET
_HomingStepZ := HomingStepX;
END_SET
END_PROPERTY

METHOD HomingX : BOOL
CASE _HomingStepX OF
		
	0:
		HomingX := FALSE;
		
		
		IF AxisX.Enable() THEN
			
			//Trace('Enable Axis X');
			_HomingStepX := _HomingStepX + 10;
		END_IF
		
	10:
		IF AxisX.Enabled THEN
			AxisX.Acceleration := 100;
			AxisX.Deceleration := 15000;
			//Trace('Enabled Axis X');
			_HomingStepX := _HomingStepX + 10;
		END_IF

	20:
		IF IO.ProximitySensorX THEN
			IF AxisX.Stop() THEN
				IF NOT AxisX.Busy THEN
				AxisX.Home();
				////Trace('Start na krańcówce X');
				_HomingStepX := 80;
				END_IF
			END_IF
		ELSE		
			_HomingStepX := _HomingStepX + 10;
		END_IF
		
	30:
		IF AxisX.MoveVelocity(-100, FALSE) THEN
			////Trace('Szybki ruch, szukam krancowki X');
            _HomingStepX := _HomingStepX + 10;
        END_IF
		
	
	40: 
		IF IO.ProximitySensorX THEN
			
		IF AxisX.Stop() THEN
			IF NOT AxisX.Busy THEN
				//Trace('Spotkałem krańcówkę X');
				_HomingStepX := _HomingStepX + 10;
			END_IF
		END_IF
		
		END_IF

	50:
		IF AxisX.MoveRelative(30,FALSE) THEN
			//Trace('Odsunięcie od krańcówki, po szybkim X');
			_HomingStepX := _HomingStepX + 10;
		END_IF
		
	60: 
		IF AxisX.MoveVelocity(-10,FALSE) THEN
			//Trace('Spokojny powrot X');		
			_HomingStepX := _HomingStepX + 10;
		END_IF	
		
	70:
		IF IO.ProximitySensorX THEN
			IF AxisX.Stop() THEN
				//Trace('Stop do precyzyjnego X');
				_HomingStepX := _HomingStepX + 10; // Przechodzimy do czekania na zatrzymanie
			END_IF
		END_IF

	80:
		IF NOT AxisX.Busy THEN
			IF AxisX.Home() THEN
				_HomingStepX := _HomingStepX + 10;
				//Trace('Precyzyjny Home wykonany X');
			END_IF
		END_IF


	90:	
		IF AxisX.MoveRelative(2.0, FALSE) THEN
			//Trace('Odsunięcie od krańcówki o 2mm X');
			_HomingStepX := _HomingStepX + 10;
		END_IF
	
	100:
		IF NOT AxisX.Busy THEN
		
			IF AxisX.Home() THEN
				//Trace('Ustawienie nowego zera po odsunięciu X');
				_HomingStepX := _HomingStepX + 10;
			END_IF
		END_IF
	
	110:
		HomingX := TRUE;
		//Trace('Homing zakończony pomyślnie X');
		
			
	END_CASE
END_METHOD

METHOD HomingY : BOOL
CASE _HomingStepY OF
		
	0:
		HomingY := FALSE;
			
		IF AxisY.Enable() THEN
			
			//Trace('Enable Axis Y');
			_HomingStepY := _HomingStepY + 10;
		END_IF
		
	10:
		IF AxisY.Enabled THEN
			AxisY.Acceleration := 100;
			AxisY.Deceleration := 15000;
			//Trace('Enabled Axis Y');
			_HomingStepY := _HomingStepY + 10;
		END_IF

	20:
		IF IO.ProximitySensorY THEN
			IF AxisY.Stop() THEN
				IF NOT AxisY.Busy THEN
				AxisY.Home();
				//Trace('Start na krańcówce Y');
				_HomingStepY := 80;
				END_IF
			END_IF
		ELSE		
			_HomingStepY := _HomingStepY + 10;
		END_IF
		
	30:
		IF AxisY.MoveVelocity(-80, FALSE) THEN
			//Trace('Szybki ruch, szukam krancowki Y');
            _HomingStepY := _HomingStepY + 10;
        END_IF
		
	
	40: 
		IF IO.ProximitySensorY THEN
			
		IF AxisY.Stop() THEN
			IF NOT AxisY.Busy THEN
				//Trace('Spotkałem krańcówkę Y');
				_HomingStepY := _HomingStepY + 10;
			END_IF
		END_IF
		
		END_IF

	50:
		IF AxisY.MoveRelative(30,FALSE) THEN
			//Trace('Odsunięcie od krańcówki, po szybkim Y');
			_HomingStepY := _HomingStepY + 10;
		END_IF
		
	60: 
		IF AxisY.MoveVelocity(-10,FALSE) THEN
			//Trace('Spokojny powrot Y');		
			_HomingStepY := _HomingStepY + 10;
		END_IF	
		
	70:
		IF IO.ProximitySensorY THEN
			IF AxisY.Stop() THEN
				//Trace('Stop do precyzyjnego Y');
				_HomingStepY := _HomingStepY + 10; // Przechodzimy do czekania na zatrzymanie
			END_IF
		END_IF

	80:
		IF NOT AxisY.Busy THEN
			IF AxisY.Home() THEN
				_HomingStepY := _HomingStepY + 10;
				//Trace('Precyzyjny Home wykonany Y');
			END_IF
		END_IF


	90:	
		IF AxisY.MoveRelative(2.0, FALSE) THEN
			//Trace('Odsunięcie od krańcówki o 2mm Y');
			_HomingStepY := _HomingStepY + 10;
		END_IF
	
	100:
		IF NOT AxisY.Busy THEN
		
			IF AxisY.Home() THEN
				//Trace('Ustawienie nowego zera po odsunięciu Y');
				_HomingStepY := _HomingStepY + 10;
			END_IF
		END_IF
	
	110:
		HomingY := TRUE;
		//Trace('Homing zakończony pomyślnie Y');
		
			
	END_CASE
END_METHOD

METHOD HomingZ : BOOL
CASE _HomingStepZ OF
		
	0:
		HomingZ := FALSE;	
		
		IF AxisZ.Enable() THEN
			
			//Trace('Enable Axis Z');
			_HomingStepZ := _HomingStepZ + 10;
		END_IF
		
	10:
		IF AxisZ.Enabled THEN
			AxisZ.Acceleration := 100;
			AxisZ.Deceleration := 15000;
			//Trace('Enabled Axis Z');
			_HomingStepZ := _HomingStepZ + 10;
		END_IF

	20:
		IF IO.ProximitySensorZ THEN
			IF AxisZ.Stop() THEN
				IF NOT AxisZ.Busy THEN
				AxisZ.Home();
				//Trace('Start na krańcówce Z');
				_HomingStepZ := 80;
				END_IF
			END_IF
		ELSE		
			_HomingStepZ := _HomingStepZ + 10;
		END_IF
		
	30:
		IF AxisZ.MoveVelocity(-100, FALSE) THEN
			//Trace('Szybki ruch, szukam krancowki Z');
            _HomingStepZ := _HomingStepZ + 10;
        END_IF
		
	
	40: 
		IF IO.ProximitySensorZ THEN
			
		IF AxisZ.Stop() THEN
			IF NOT AxisZ.Busy THEN
				//Trace('Spotkałem krańcówkę Z');
				_HomingStepZ := _HomingStepZ + 10;
			END_IF
		END_IF
		
		END_IF

	50:
		IF AxisZ.MoveRelative(5,FALSE) THEN
			//Trace('Odsunięcie od krańcówki, po szybkim Z');
			_HomingStepZ := _HomingStepZ + 10;
		END_IF
		
	60: 
		IF AxisZ.MoveVelocity(-10,FALSE) THEN
			//Trace('Spokojny powrot Z');		
			_HomingStepZ := _HomingStepZ + 10;
		END_IF	
		
	70:
		IF IO.ProximitySensorZ THEN
			IF AxisZ.Stop() THEN
				//Trace('Stop do precyzyjnego Z');
				_HomingStepZ := _HomingStepZ + 10; // Przechodzimy do czekania na zatrzymanie
			END_IF
		END_IF

	80:
		IF NOT AxisZ.Busy THEN
			IF AxisZ.Home() THEN
				_HomingStepZ := _HomingStepZ + 10;
				//Trace('Precyzyjny Home wykonany Z');
			END_IF
		END_IF


	90:	
		IF AxisZ.MoveRelative(2.0, FALSE) THEN
			//Trace('Odsunięcie od krańcówki o 2mm Z');
			_HomingStepZ := _HomingStepZ + 10;
		END_IF
	
	100:
		IF NOT AxisZ.Busy THEN		
		
			IF AxisZ.Home() THEN
				//Trace('Ustawienie nowego zera po odsunięciu Z');
				_HomingStepZ := _HomingStepZ + 10;
			END_IF
		END_IF
	
	110:
		HomingZ := TRUE;
		//Trace('Homing zakończony pomyślnie Z');
		
			
	END_CASE
END_METHOD

//! @summary Basic module initialization logic
METHOD PROTECTED Initialize : BOOL;
VAR
    i                        : UDINT;
    varInfo                  : __SYSTEM.VAR_INFO;
    AllSubUnitsInitialized   : BOOL := TRUE;
    AllComponentsInitialized : BOOL := TRUE;
END_VAR

//! @description This method is called by <c>CyclicLogic()</c> as required
Initialize := FALSE;
CASE DescendantSequenceState OF
    0:
		RegisterComponent(AxisX);
		RegisterComponent(AxisY);	
		RegisterComponent(AxisZ);	
		RegisterComponent(CylinderCuttingY);
		RegisterComponent(CylinderCuttingX);
        _LogModeChanges         := FALSE;
        _LogStateChanges        := FALSE;
        DescendantSequenceState := DescendantSequenceState + 10;
    10:
		IF RestorePersistentData() THEN
		
		// Przypisanie osi do strategii
		fbHomeStratX.Axis := AxisX;
		fbHomeStratY.Axis := AxisY;
		fbHomeStratZ.Axis := AxisZ;
		
		// Wstrzyknięcie strategii do osi (Dependency Injection)
		AxisX.HomeMethod := fbHomeStratX;
		AxisY.HomeMethod := fbHomeStratY;
		AxisZ.HomeMethod := fbHomeStratZ;
		
		
        DescendantSequenceState := DescendantSequenceState + 10;
		//initialize persistent
		END_IF
    20:
        //Copy Mode names
        FOR i := 1 TO 3 DO
            ModeNames[i] := F_UnitModeToString(UDINT_TO_DINT(i));
        END_FOR

        DescendantSequenceState := DescendantSequenceState + 10;
    30:
        //Call the Super
        IF SUPER^.Initialize() THEN
            DescendantSequenceState := DescendantSequenceState + 10;
        END_IF
    40:
        Initialize := TRUE;
END_CASE
END_METHOD

METHOD MachiningOrchestrator : BOOL
VAR_INST
		Timer			:TON;
END_VAR
CASE OrchestratorStep OF
    0: // Enable osi
        
        OrchestratorStep := 5;
      

    5: // Zbuduj odcinki dla tego programu
				CASE _ProgramIdRequested OF
					
					E_RecipeID.eBorgoFlaps:
					IF BuildSegments_BorgoFlaps() THEN
						OrchestratorStep := OrchestratorStep + 10;
					END_IF
					
					E_RecipeID.eBorgoWings:
					IF BuildSegments_BorgoWings() THEN
						OrchestratorStep := OrchestratorStep + 10;
					END_IF
					
					E_RecipeID.eArona:
					IF BuildSegments_Arona() THEN
						OrchestratorStep := OrchestratorStep + 10;
					END_IF
					
				END_CASE        

        OrchestratorStep := 10;

    10: 
        IF ExecuteSegmentsGroove() THEN
           OrchestratorStep := 20;
        END_IF
		
	20: 
	 	IF ExecuteSegmentsCutY() THEN
            OrchestratorStep := 30;
        END_IF
		
	30: 
	 	IF ExecuteSegmentsCutX() THEN
            OrchestratorStep := 40;
        END_IF	

    40:
        IF AxisZ.InPosition AND AxisX.InPosition AND AxisY.InPosition THEN
            MachiningOrchestrator := TRUE;
        END_IF
END_CASE
END_METHOD

PROPERTY PUBLIC PanelFrontWidth : REAL
GET
PanelFrontWidth := _PanelFrontWidth;
END_GET
SET
_PanelFrontWidth := PanelFrontWidth;
END_SET
END_PROPERTY

PROPERTY PUBLIC PanelHeight : REAL
GET
PanelHeight := _PanelHeight;
END_GET
SET
_PanelHeight := PanelHeight;
END_SET
END_PROPERTY

PROPERTY ProgramIdRequested : E_RecipeID
GET
ProgramIdRequested := _ProgramIdRequested;
END_GET
SET
_ProgramIdRequested := ProgramIdRequested;
END_SET
END_PROPERTY

PROPERTY PUBLIC RailHeightCorrection : REAL
GET
RailHeightCorrection := _RailHeightCorrection;
END_GET
SET
 IF RailHeightCorrection > 15 THEN
	_RailHeightCorrection := 15;  // It can't go higher, you will kill yourself
	ELSE
	_RailHeightCorrection := RailHeightCorrection;
END_IF
END_SET
END_PROPERTY

PROPERTY PUBLIC RapidSpeedX : REAL
GET
RapidSpeedX := _RapidSpeedX;
END_GET
SET
_RapidSpeedX := RapidSpeedX;
END_SET
END_PROPERTY

PROPERTY PUBLIC RapidSpeedY : REAL
GET
RapidSpeedY := _RapidSpeedY;
END_GET
SET
_RapidSpeedY := RapidSpeedY;
END_SET
END_PROPERTY

PROPERTY PUBLIC RapidSpeedZ : REAL
GET
RapidSpeedZ := _RapidSpeedZ;
END_GET
SET
_RapidSpeedZ := RapidSpeedZ;
END_SET
END_PROPERTY

METHOD ResetSafety : BOOL
VAR_INST
	Step : INT ;	
	SafetyTimer :TON;
	SafetyTimerTrigger :R_TRIG;
END_VAR
//auto resetting timer, a start condition is an end condition
SafetyTimer(IN:= Step > 0 AND NOT SafetyTimer.Q, PT:= T#500MS);

CASE Step OF
		
		0:  // Reset group or waits
			ResetSafety:= FALSE;
			Trace('Timer Initialize');
			Step := Step + 10;
			
		10: //If necessary reset group
		
			GVL_Safety.ErrorAck := (GVL_Safety.ComError OR GVL_Safety.FBError); 
		
			IF GVL_Safety.ErrorAck OR SafetyTimer.Q THEN 
				Step := Step + 10;
			END_IF

		20: //Wait for the signal propagation
			IF SafetyTimer.Q THEN
				GVL_Safety.ErrorAck := FALSE;
				Step := Step + 10;
			END_IF
		
		30: //Check FB errors
			IF GVL_Safety.FBError OR (NOT GVL_Safety.SafetyPermission) THEN
				GVL_Safety.RestartFBs := TRUE;
			END_IF
			
			Step := Step + 10;
			
		40: //Wait for the signal propagation
		
			IF SafetyTimer.Q THEN
				GVL_Safety.RestartFBs := FALSE;
				Step := Step + 10;
			END_IF	
			
		50: //Wait for the signal propagation
			
			
		IF SafetyTimer.Q THEN
				
			
				IF GVL_Safety.SafetyPermission AND 
					NOT (GVL_Safety.ComError OR GVL_Safety.FBError OR GVL_Safety.SafeError) 
				
					THEN
						Step := 0;
						ResetSafety := TRUE;
					ELSE
						Step := 0;
						ResetSafety := FALSE;
				END_IF
			
			END_IF
		
		ELSE
		
		Step := 0;	

END_CASE
END_METHOD

METHOD PROTECTED Resetting
VAR
	i				: UDINT;
	SubModulesReady : BOOL := TRUE;
	

	
END_VAR

VAR_INST
	flagX :BOOL;
	flagY :BOOL;
	flagZ :BOOL;
END_VAR
CASE _CurrentMode OF

	//=================================PRODUCTION MODE==================================
	E_PMLUnitMode.ePMLUnitMode_Production:
		CASE SequenceState OF
			0:
				NoStateTasksToComplete := FALSE;
				SequenceState := SequenceState + 5;


			5:

				AxisX.WriteParameter(MC_AxisParameter.AxisMinSoftPosLimit, -1250);	 
				AxisX.WriteParameter(MC_AxisParameter.AxisMaxSoftPosLimit, 1250);
		
				AxisY.WriteParameter(MC_AxisParameter.AxisMinSoftPosLimit, -2300);	 
				AxisY.WriteParameter(MC_AxisParameter.AxisMaxSoftPosLimit, 2300);
		
				AxisZ.WriteParameter(MC_AxisParameter.AxisMinSoftPosLimit, -100);	 
				AxisZ.WriteParameter(MC_AxisParameter.AxisMaxSoftPosLimit, 100);	
				
				SequenceState := SequenceState + 5;
		
			10: 
      			
			  AxisX.Enable();
			  AxisY.Enable();
			  AxisZ.Enable();
	 
			SequenceState := 12;
		
		12:
        
        // 2. Czekamy, aż napędy "wstaną" i zameldują gotowość
        IF AxisX.Enabled AND AxisY.Enabled AND AxisZ.Enabled THEN
            SequenceState := 15;
        END_IF
        
15:
        // 1. "Bombardujemy" osie komendami, dopóki każda z osobna nie odpowie TRUE
        IF NOT flagX THEN flagX := AxisX.Home(); END_IF
        IF NOT flagY THEN flagY := AxisY.Home(); END_IF
        IF NOT flagZ THEN flagZ := AxisZ.Home(); END_IF

        // 2. Kiedy cała trójka potwierdziła przyjęcie rozkazu:
        IF flagX AND flagY AND flagZ THEN
            // Czyścimy flagi przed następnym użyciem maszyny!
            flagX := FALSE;
            flagY := FALSE;
            flagZ := FALSE;
            
            SequenceState := 20; // Idziemy czekać na koniec ruchu
        END_IF
					
	20:			
//			IF AxisX.Axis.Status.Homed AND AxisY.Axis.Status.Homed AND AxisZ.Axis.Status.Homed THEN
			IF AxisX.Axis.Status.Homed AND AxisY.Axis.Status.Homed AND AxisZ.Axis.Status.Homed THEN
//			IF flagX AND flagY AND flagZ THEN

				Trace('All Axes Homing completed');
				flagX :=0; 
				flagY :=0; 
				flagZ :=0;
				OrchestratorStep := 0;
				ExecutorStep := 0;
				THIS^.HomingStepX := 0;
				THIS^.HomingStepY := 0;
				THIS^.HomingStepZ := 0;
				SequenceState := 40;
//			END_IF			
			END_IF		
			40:		
				StateTasksComplete := TRUE;
				SUPER^.Resetting();
		END_CASE

	//=================================MAINTENANCE & MANUAL MODE==================================
	E_PMLUnitMode.ePMLUnitMode_Maintenance:

	CASE SequenceState OF
			0:
				NoStateTasksToComplete := FALSE;
				SequenceState := SequenceState + 10;	
		
			10: 
				AxisX.Enable();
				AxisY.Enable();
				AxisZ.Enable();	
				
				IF AxisX.Enabled AND AxisY.Enabled AND AxisZ.Enabled THEN
					SequenceState := SequenceState + 10;
				END_IF
				
			20:	

				AxisX.WriteParameter(MC_AxisParameter.AxisMinSoftPosLimit, -1250);	 
				AxisX.WriteParameter(MC_AxisParameter.AxisMaxSoftPosLimit, 1250);
		
				AxisY.WriteParameter(MC_AxisParameter.AxisMinSoftPosLimit, -2300);	 
				AxisY.WriteParameter(MC_AxisParameter.AxisMaxSoftPosLimit, 2300);
		
				AxisZ.WriteParameter(MC_AxisParameter.AxisMinSoftPosLimit, -100);	 
				AxisZ.WriteParameter(MC_AxisParameter.AxisMaxSoftPosLimit, 100);
			
				SequenceState := SequenceState + 10;
			30:
	
				SequenceState := SequenceState + 10;
					
			40:		
				StateTasksComplete := TRUE;
				SUPER^.Resetting();
		END_CASE
	
 	E_PMLUnitMode.ePMLUnitMode_Manual:
			
	CASE SequenceState OF
			0:
				NoStateTasksToComplete := FALSE;
				SequenceState := SequenceState + 10;	
		
			10: 
				AxisX.Enable();
				AxisY.Enable();
				AxisZ.Enable();	
				
				IF AxisX.Enabled AND AxisY.Enabled AND AxisZ.Enabled THEN
					SequenceState := SequenceState + 10;
				END_IF
				
			20:	

				AxisX.WriteParameter(MC_AxisParameter.AxisMinSoftPosLimit, -1250);	 
				AxisX.WriteParameter(MC_AxisParameter.AxisMaxSoftPosLimit, 1250);
		
				AxisY.WriteParameter(MC_AxisParameter.AxisMinSoftPosLimit, -2300);	 
				AxisY.WriteParameter(MC_AxisParameter.AxisMaxSoftPosLimit, 2300);
		
				AxisZ.WriteParameter(MC_AxisParameter.AxisMinSoftPosLimit, -100);	 
				AxisZ.WriteParameter(MC_AxisParameter.AxisMaxSoftPosLimit, 100);
			
				SequenceState := SequenceState + 10;
			30:
	
				SequenceState := SequenceState + 10;
					
			40:		
				StateTasksComplete := TRUE;
				SUPER^.Resetting();
		END_CASE
		
	
	END_CASE
END_METHOD

METHOD RestorePersistentData : BOOL
//Only _Variables are PERSISTENT, This method is executed during the initialization

GantryXYZ_HMI.Config.CutterXOffsetX       := _CutterXOffsetX;
GantryXYZ_HMI.Config.CutterXOffsetY       := _CutterXOffsetY;
GantryXYZ_HMI.Config.CutterYOffsetX       := _CutterYOffsetX;
GantryXYZ_HMI.Config.CutterYOffsetY       := _CutterYOffsetY;
GantryXYZ_HMI.Config.CuttingSpeedX        := _CuttingSpeedX;
GantryXYZ_HMI.Config.CuttingSpeedY        := _CuttingSpeedY;
GantryXYZ_HMI.Config.CuttingIdleTime      := _CuttingIdleTime;
GantryXYZ_HMI.Config.CuttingOverpass      := _CuttingOverpass;
GantryXYZ_HMI.Config.GrooveDepthZ         := _GrooveDepthZ;
GantryXYZ_HMI.Config.GroovingSpeedX       := _GroovingSpeedX;
GantryXYZ_HMI.Config.GroovingSpeedY       := _GroovingSpeedY;
GantryXYZ_HMI.Config.GroovingSpeedZ       := _GroovingSpeedZ;
GantryXYZ_HMI.Config.GroovingIdleTime     := _GroovingIdleTime;
GantryXYZ_HMI.Config.GroovingOverpass     := _GroovingOverpass;
GantryXYZ_HMI.Config.RapidSpeedX          := _RapidSpeedX;
GantryXYZ_HMI.Config.RapidSpeedY          := _RapidSpeedY;
GantryXYZ_HMI.Config.RapidSpeedZ          := _RapidSpeedZ;
GantryXYZ_HMI.Config.GlobalOffset		  := _GlobalOffset;

//GantryXYZ_HMI.Config.PanelFrontLength     := _PanelFrontLength;
GantryXYZ_HMI.Config.PanelFrontWidht      := _PanelFrontWidth;
GantryXYZ_HMI.Config.PanelHeight          := _PanelHeight;
GantryXYZ_HMI.Config.RailHeightCorrection := _RailHeightCorrection;


RestorePersistentData := TRUE;
END_METHOD

METHOD SequenceTimerSeconds : BOOL
VAR_INPUT
	WaitingTime :REAL;
END_VAR

VAR_INST
	 Timer :TON;
END_VAR
 Timer(IN := TRUE, PT := REAL_TO_TIME(WaitingTime * 1000.0));
 IF Timer.Q THEN
	Timer(IN := FALSE);
	SequenceTimerSeconds := TRUE;
END_IF
END_METHOD

END_FUNCTION_BLOCK

(* stored: Version 1.1.0.1, ProductVersion 3.1.4024.15
   POU FB_GantryXYZ: Id {474e1990-f731-0ed9-052c-42626742a38f}, SpecialFunc None
   Folder MyMethods: Id {d166ca9d-f57a-4d88-ac90-142e5eb5d488}
   Folder Segments: Id {b8033ee7-c5f7-43d2-a584-12e2969c60b8}
   Folder Properties: Id {b05cc7e1-dc37-4910-986a-f085b4a0163d}
   Folder Comand: Id {afdb6df3-76c4-47c1-997d-636ee1fa8ab3}
   Folder Config: Id {d432f26c-f18e-459c-b74b-59233683f472}
   Folder Status: Id {76f95e74-5bed-4ec3-be3e-2b7b97f61740}
   Folder States: Id {8df42c9b-c051-49f1-9767-900503632339}
   Method Aborting: Id {5476dfef-6652-4e6b-8928-3724a50553de}
   Method BuildSegments_Arona: Id {e84aaa35-d3d2-459f-b6b9-b01f1c51048b}
   Method BuildSegments_BorgoFlaps: Id {30aff943-63a2-49df-9f71-8b8f78deda49}
   Method BuildSegments_BorgoWings: Id {0600b631-5666-4473-9115-8ec263b291bb}
   Method BuildSegments_Calibration: Id {0bc1bcc0-1e48-4916-b44b-21d9143ba598}
   Method Clearing: Id {9be5800b-bdc3-471f-9b7d-42ef121d5c77}
   Method Completing: Id {6c861ff6-52ea-4daf-b956-f189ed9d190d}
   Method CreateEvents: Id {40e5a283-7f33-033f-0879-cc11ecabc43d}
   Property CurrentSpeed: Id {357ae8db-7056-4092-8dce-8465b738ac10}
   Get Get: Id {c2cd3b04-3efb-4ba6-9575-51c55bf7cfdf}
   Property CutterXOffsetX: Id {ec876c40-72b1-49ef-b4a8-dafc4e3faf39}
   Get Get: Id {84da6823-a94d-424f-a88e-9f4900452f7f}
   Set Set: Id {415034c5-edcb-4d81-8764-a7aa31c1615f}
   Property CutterXOffsetY: Id {195bbbbb-15a8-436d-866c-ecc00711e6f4}
   Get Get: Id {c99ef4e3-05c1-488d-a09a-ef00fdd76f8d}
   Set Set: Id {dfc0ea26-14ea-4173-aef3-e2791575f96a}
   Property CutterYOffsetX: Id {2d729998-2abb-43f8-849d-8b6a18e55ff7}
   Get Get: Id {dd957d56-9ca4-4d71-901a-4eee0dcc7dcb}
   Set Set: Id {8614b2fc-b567-4793-b660-6be46ebcc9c1}
   Property CutterYOffsetY: Id {f510443c-1bf0-4520-86a8-c58e1e7a4692}
   Get Get: Id {0ec517ed-6f75-4191-aed5-4585f3f07608}
   Set Set: Id {a114f71c-22b7-478b-aa78-245d801668e5}
   Property CuttingIdleTime: Id {61054465-d4b7-49c6-8b84-c09fde09dffb}
   Get Get: Id {fd9fc4d0-2df8-4834-aea2-4450714f930b}
   Set Set: Id {b29e1f37-0d7e-428c-a22d-0afaabad6d2b}
   Property CuttingOverpass: Id {b1a537b6-c123-47df-9f6b-c4bd2f95e73a}
   Get Get: Id {257c3c0a-0042-41f3-b22c-f718e636d2ad}
   Set Set: Id {93b54848-7c11-4e5b-9e28-1fa78fa03fbc}
   Property CuttingSpeedX: Id {12a88485-b295-4495-a76e-0eceef2a24df}
   Get Get: Id {e7a4474f-22fa-456b-9710-abf007c43654}
   Set Set: Id {41d1285e-069d-4d01-b574-3be12c525491}
   Property CuttingSpeedY: Id {9e82d40a-2e51-4b4a-b71e-9294ce0c8388}
   Get Get: Id {bfc37d4f-4d55-4a0f-beca-3b432877e9ac}
   Set Set: Id {58519851-d00e-4316-b0a9-8db16980a7cd}
   Method CyclicLogic: Id {0cfbfa67-40d6-05d6-0515-ef1c50353a78}
   Method Execute: Id {895d1ef9-5e85-47dd-a8bf-b32885837641}
   Method ExecuteSegmentsCutX: Id {94347c53-d843-4c0f-8fa0-b761cd0d80e2}
   Method ExecuteSegmentsCutY: Id {dc7ba1fd-c66f-4871-a334-3c135aa8a2cb}
   Method ExecuteSegmentsGroove: Id {3ee66abc-6845-49e5-b2ff-149134d7252b}
   Property GlobalOffset: Id {c8ddd37c-b19a-4d4e-a71b-b97d8605e766}
   Get Get: Id {688e3d94-1410-4383-b142-64e21d43f1a6}
   Set Set: Id {5f121375-3c35-4dc4-9401-8a845e0cf0c0}
   Property GrooveDepthZ: Id {4c86fbb5-f7fe-4ab0-abb5-4601fd04a1c4}
   Get Get: Id {a83b65c4-5ea3-488c-967b-3ee17e2e67f9}
   Set Set: Id {3fde4dcd-fcc8-4a85-8a9a-5adb0df55581}
   Property GroovingIdleTime: Id {dfb103a6-b180-49ba-a124-4e96d3059088}
   Get Get: Id {d6ada8f0-07b8-4d16-9743-4e216d422b6a}
   Set Set: Id {e8df0304-5562-4c08-bd77-ccab9fffa15b}
   Property GroovingOverpass: Id {812d4990-d277-4bfc-8e06-a4ff70191e9b}
   Get Get: Id {b0c9f572-3145-4e3a-b91c-cd20c9ba4da8}
   Set Set: Id {826fd5bf-1fa9-4f64-9665-346b4d89d6bf}
   Property GroovingSpeedX: Id {ab870480-cf07-40c0-bfcb-dd69cb432ee7}
   Get Get: Id {6314d467-3274-40d3-b79c-da2e9e92d14f}
   Set Set: Id {187fbc7b-15d7-49b2-9b45-3a42d4ac6f21}
   Property GroovingSpeedY: Id {dbf5c766-18d1-470a-99da-17fb86de0bc4}
   Get Get: Id {857e501f-f2f5-4e77-9eae-4cbc8957979e}
   Set Set: Id {e1f697d5-7820-41ea-a263-d25f9b120395}
   Property GroovingSpeedZ: Id {1df46c0c-e665-451c-ba3a-e7e742b71643}
   Get Get: Id {bacd8e8f-7f73-4606-b74b-5e23e6d6dcf2}
   Set Set: Id {dea83ede-69cc-4213-8244-a1bc2a541f42}
   Method HMICommunication: Id {0dce72f4-da14-4dd2-b6a3-5db9db3404e0}
   Method HMIPermissions: Id {a7a517c4-9176-4ef6-9045-d889c05c8a21}
   Property HomingStepX: Id {bb0ed88a-091c-4bab-9e01-a967ca1fc9bb}
   Get Get: Id {190b2c1a-84a4-4b9a-b82b-d034c6e97b13}
   Set Set: Id {9c9687a4-cd61-4104-a02f-3fe4715cd2fa}
   Property HomingStepY: Id {b85ccf6c-14f7-4091-9161-3a64d81c6f71}
   Get Get: Id {c9fc6e3e-e251-4188-a708-1d897bfbe015}
   Set Set: Id {51c79bd9-40f7-4370-9e3f-edffa2a24928}
   Property HomingStepZ: Id {0b9a390e-db9e-4739-bffa-5ca069d437ef}
   Get Get: Id {403aef28-5a6c-4ea4-b639-a6922b7be29b}
   Set Set: Id {5b912885-4f7d-414a-b1af-1074244e821d}
   Method HomingX: Id {3a7dd60d-4e3b-4739-b0ec-f4ab527c9236}
   Method HomingY: Id {7cf726af-0fa2-4719-9f55-f55ebcdc06af}
   Method HomingZ: Id {59c5c153-dee1-4d97-aac8-e655f142ebf1}
   Method Initialize: Id {ba85f303-ffbe-03ad-229b-3741bd93e6e2}
   Method MachiningOrchestrator: Id {4a6c8d9d-4b5c-46da-8179-e7275fa91b7f}
   Property PanelFrontWidth: Id {f3e0dbc8-c3fa-460e-86ce-eb87111125e9}
   Get Get: Id {337b7ccf-7529-41b1-81a1-e9c0f98de875}
   Set Set: Id {6f7f0fd9-fb5c-4077-ab43-02d47a14a15f}
   Property PanelHeight: Id {0920acc0-257a-43b2-a196-f22fc89e42ed}
   Get Get: Id {20b3fa55-de19-44e2-ad7b-52463e1bf19b}
   Set Set: Id {91d58d60-235c-48ff-9b62-1155794955c4}
   Property ProgramIdRequested: Id {3b163a54-6fcd-4be2-bb98-ad529d342348}
   Get Get: Id {21210547-61ea-4bd8-a78a-96552b4742ab}
   Set Set: Id {2bb8002c-0857-45bb-b53e-f611a5c233b9}
   Property RailHeightCorrection: Id {465e1c57-83b8-4b2a-a3fe-16819241fd4f}
   Get Get: Id {8547e8a4-2368-4b1c-bac1-a9f1330a50a7}
   Set Set: Id {77d9b924-4d53-4d00-8d3d-e32bf531a5d3}
   Property RapidSpeedX: Id {8c9f4f21-3743-48de-8aa6-1e7f68956f80}
   Get Get: Id {80bdcbb9-4e80-4343-9582-3dba51122fa5}
   Set Set: Id {5ccad6ef-816c-4c49-afb6-3e5204fc4fb5}
   Property RapidSpeedY: Id {5dfea665-2261-44a4-b000-9743b481b2b9}
   Get Get: Id {59b145df-2cff-4ecc-847b-f8d110514f0e}
   Set Set: Id {4f8d9cc9-05ef-4eb8-8eb1-49992a2bb0d6}
   Property RapidSpeedZ: Id {cebf8cd2-acc1-4736-8c92-219e5578dd1a}
   Get Get: Id {11b4159d-524a-4e2d-b881-810c4516a42c}
   Set Set: Id {e54cbdaf-56e9-49ed-85a4-52a0db9e7c8e}
   Method ResetSafety: Id {6bac4035-16f4-4bf2-95a7-9f0b204a82b7}
   Method Resetting: Id {e7a01217-de28-430f-aeef-f83d9f1b6f0d}
   Method RestorePersistentData: Id {9e1193e7-d277-4fd9-ac0c-81f097451afd}
   Method SequenceTimerSeconds: Id {2e721ea1-cfa0-448e-b2fb-baa077a6b9b3} *)
